FUNCTION_BLOCK TcoSingleAxisPositionsRootContainer EXTENDS TcoCore.TcoObject
VAR_INPUT
END_VAR
VAR_OUTPUT
END_VAR
VAR
END_VAR

END_FUNCTION_BLOCK

(* stored: Version 1.1.0.1, ProductVersion 3.1.4024.12
   POU TcoSingleAxisPositionsRootContainer: Id {9450a862-e6ad-0399-1428-c975950add9f}, SpecialFunc None *)
